INTERFACE I_RecipeBuilder

PROPERTY ActualCopiesX : DINT
GET
END_GET
END_PROPERTY

PROPERTY ActualCopiesY : DINT
GET
END_GET
END_PROPERTY

METHOD Build : BOOL
END_METHOD

PROPERTY Busy : BOOL
GET
END_GET
SET
END_SET
END_PROPERTY

PROPERTY Config : ST_RecipeBuilder_Config
GET
END_GET
SET
END_SET
END_PROPERTY

PROPERTY ConfigProvider : I_GantryConfigProvider
GET
END_GET
SET
END_SET
END_PROPERTY

PROPERTY Done : BOOL
GET
END_GET
SET
END_SET
END_PROPERTY

PROPERTY Error : BOOL
GET
END_GET
SET
END_SET
END_PROPERTY

PROPERTY ExecutionRoute : E_ExecutionRoute
GET
END_GET
END_PROPERTY

PROPERTY FootprintX : REAL
GET
END_GET
SET
END_SET
END_PROPERTY

PROPERTY FootprintY : REAL
GET
END_GET
SET
END_SET
END_PROPERTY

PROPERTY GeometryWriter : I_GeometryWriter
GET
END_GET
SET
END_SET
END_PROPERTY

PROPERTY HolesDrill : REFERENCE TO ARRAY [1..32] OF ST_PointXY;
GET
END_GET
END_PROPERTY

PROPERTY HolesToDrill : INT
GET
END_GET
END_PROPERTY

PROPERTY Limits : ST_Recipe_Limits
GET
END_GET
END_PROPERTY

PROPERTY MaxCopiesX : DINT
GET
END_GET
END_PROPERTY

PROPERTY MaxCopiesY : DINT
GET
END_GET
END_PROPERTY

PROPERTY SegmentsCutX : REFERENCE TO ARRAY [1..32] OF ST_CutSegment
GET
END_GET
END_PROPERTY

PROPERTY SegmentsCutY : REFERENCE TO ARRAY [1..32] OF ST_CutSegment
GET
END_GET
END_PROPERTY

PROPERTY SegmentsGroove : REFERENCE TO ARRAY [1..32] OF ST_CutSegment
GET
END_GET
END_PROPERTY

PROPERTY SegmentsToCutX : INT
GET
END_GET
END_PROPERTY

PROPERTY SegmentsToCutY : INT
GET
END_GET
END_PROPERTY

PROPERTY SegmentsToGroove : INT
GET
END_GET
END_PROPERTY

END_INTERFACE

(* stored: Version 1.1.0.1, ProductVersion 3.1.4024.15
   Itf I_RecipeBuilder: Id {a1b2c3d4-1111-4222-b333-c4d5e6f7a8b9}
   Property ActualCopiesX: Id {93f98e6b-9908-4fa8-90b8-6d20c29c4d3d}
   Get Get: Id {86d8b705-994d-4916-92a6-238c5db62e3d}
   Property ActualCopiesY: Id {7e141ee8-6e54-4135-beeb-8538b9a6f573}
   Get Get: Id {2f0ec9ec-a180-44b4-8a35-98706e68099d}
   Method Build: Id {b2c3d4e5-2222-4333-c444-d5e6f7a8b9c0}
   Property Busy: Id {b05530b6-09cc-4522-af33-84f83497b22f}
   Get Get: Id {56984f1d-bedb-40d9-a933-bdb8e55d91ce}
   Set Set: Id {97956bca-fc96-45f4-9b2d-26a34a9f1cc3}
   Property Config: Id {41a1f94d-1ba6-473a-8fd2-d71e6a5c7ac8}
   Get Get: Id {9b92c909-482e-45d4-839d-e73654fca949}
   Set Set: Id {e3c0a41f-b8d2-4dbf-bb3c-74c7ca0bddef}
   Property ConfigProvider: Id {d69d8d19-57dd-41af-92cc-1dbb43000e55}
   Get Get: Id {0f75a252-3e55-499a-815d-f787c9ce2267}
   Set Set: Id {db2e7971-1ba6-4a42-8104-1c956218d8fa}
   Property Done: Id {e09b3c59-4d66-4bec-b5f8-a0864915d785}
   Get Get: Id {2fe5a509-c50d-4bcd-96cf-e3705a06840a}
   Set Set: Id {699a33eb-4116-4960-9278-9781a6101fdb}
   Property Error: Id {1e30a85a-1302-494a-ac13-0c5613db912a}
   Get Get: Id {d93d9f60-85e7-4a7e-88b1-6c269c18fcfc}
   Set Set: Id {5f69266e-4525-4da8-91b5-725368d3751b}
   Property ExecutionRoute: Id {961feff0-1b35-44a7-a40f-aa8e8218ab76}
   Get Get: Id {0600c360-f7b0-4067-a18f-ab3f6a6a02ac}
   Property FootprintX: Id {b2c0660e-2273-4d0b-a3ff-b3d685a837ce}
   Get Get: Id {1c249b0f-2c24-4249-828f-a42f5a98a347}
   Set Set: Id {69901a39-3c4a-43c9-9774-7abb6f456824}
   Property FootprintY: Id {2613b715-d424-4985-974e-570c5f3a3a3a}
   Get Get: Id {0c30c23d-b3d9-441f-89eb-313480456f50}
   Set Set: Id {0a3a18d1-13c3-4727-bb69-a7fa42e8a244}
   Property GeometryWriter: Id {d4bebd77-571d-4217-889b-872c8fc3a75b}
   Get Get: Id {d6a12bab-d176-4870-bbae-066a355dfdd1}
   Set Set: Id {36c32498-a83b-42dd-8e8e-4ca52f21093a}
   Property HolesDrill: Id {444fc5fe-9152-4ad9-900c-81717334843f}
   Get Get: Id {f77b18ec-e030-4941-a5d0-463fd5ae46b3}
   Property HolesToDrill: Id {00dcb715-64ce-492e-9e67-b50c838c1693}
   Get Get: Id {90bf7f9c-2a31-4ed8-8928-88c7f9f98356}
   Property Limits: Id {cb52d8bb-7c49-4fc2-8442-7c9db617c87d}
   Get Get: Id {b51051d6-7967-4941-b388-23830aee7422}
   Property MaxCopiesX: Id {80561300-5824-4fdd-b673-c3b63715f9cc}
   Get Get: Id {c3b2298d-4a22-4272-b922-207a37d98bca}
   Property MaxCopiesY: Id {3d171b71-8d34-4596-a820-b575dcc06d2f}
   Get Get: Id {e36b60ee-0613-460f-b3fe-fc821a59a2b1}
   Property SegmentsCutX: Id {a7b8c9d0-7777-4888-b999-c0d1e2f3a4b5}
   Get Get: Id {b8c9d0e1-8888-4999-c000-d1e2f3a4b5c6}
   Property SegmentsCutY: Id {e1f2a3b4-bbbb-4ccc-f333-a4b5c6d7e8f9}
   Get Get: Id {f2a3b4c5-cccc-4ddd-a444-b5c6d7e8f9a0}
   Property SegmentsGroove: Id {c3d4e5f6-3333-4444-d555-e6f7a8b9c0d1}
   Get Get: Id {d4e5f6a7-4444-4555-e666-f7a8b9c0d1e2}
   Property SegmentsToCutX: Id {c9d0e1f2-9999-4aaa-d111-e2f3a4b5c6d7}
   Get Get: Id {d0e1f2a3-aaaa-4bbb-e222-f3a4b5c6d7e8}
   Property SegmentsToCutY: Id {a3b4c5d6-dddd-4eee-b555-c6d7e8f9a0b1}
   Get Get: Id {b4c5d6e7-eeee-4fff-c666-d7e8f9a0b1c2}
   Property SegmentsToGroove: Id {e5f6a7b8-5555-4666-f777-a8b9c0d1e2f3}
   Get Get: Id {f6a7b8c9-6666-4777-a888-b9c0d1e2f3a4} *)
